{attribute addProperty BoxType "AT2050-0500-0019"}
{attribute addProperty Id "A_0094_AT2021_5250_0018_AT2021_5250AT2021_3DCFC8D064080"}
{attribute addProperty CRC "385656825"}
{attribute addProperty SizeInBites "640"}
{attribute addProperty SizeInBytes "80"}
TYPE A_0050_AT2050_0500_0019_16FCA7F9 EXTENDS AT2050_9506A482 :
STRUCT
	{attribute addProperty Name "A_0094_AT2021_5250_0018_AT2021_5250"}
	A_0094_AT2021_5250_0018_AT2021_5250 : AT2021_3DCFC8D0;
END_STRUCT
END_TYPE

(* stored: Version 1.2.0.0, ProductVersion 3.1.4024.9
   DUT A_0050_AT2050_0500_0019_16FCA7F9: Id {64fd9d74-365a-44cc-8eab-ec0174e9494f} *)
